// TIA Portal V17 export
// export: Created 2025-01-08T13:55:31.8080412Z, ExportSetting WithDefaults, DisplayName Totally Integrated Automation Portal, DisplayVersion V17, DisplayName TIA Portal Openness, DisplayVersion V17, DisplayName TIA Portal Version Control Interface, DisplayVersion V17, DisplayName SINAMICS Startdrive Advanced, DisplayVersion V17 Update2, DisplayName SINAMICS Startdrive G130, G150, S120, S150, SINAMICS MV, S210, DisplayVersion V17 Update2, DisplayName SINAMICS Startdrive G110M, G120, G120C, G120D, G120P, G115D, DisplayVersion V17 Update2, DisplayName STEP 7 Professional, DisplayVersion V17, DisplayName STEP 7 Safety, DisplayVersion V17, DisplayName WinCC Advanced, DisplayVersion V17
FUNCTION_BLOCK "FB_Com"   // FB1, LAD
{ S7_Optimized_Access := 'TRUE' }
VERSION : 0.1
// stored: AutoNumber true, IsIECCheckEnabled false, IsRetainMemResEnabled false, MemoryReserve 100, SetENOAutomatically false, UDAEnableTagReadback false
   VAR
      TRCV_C_Instance { S7_SetPoint := 'True'} : TRCV_C;
      GET_Instance { S7_SetPoint := 'True'} : GET;
      TRCV_C_Instance_1 { S7_SetPoint := 'True'} : TRCV_C;
      Diff : LInt;
   END_VAR
BEGIN

REGION Network 1
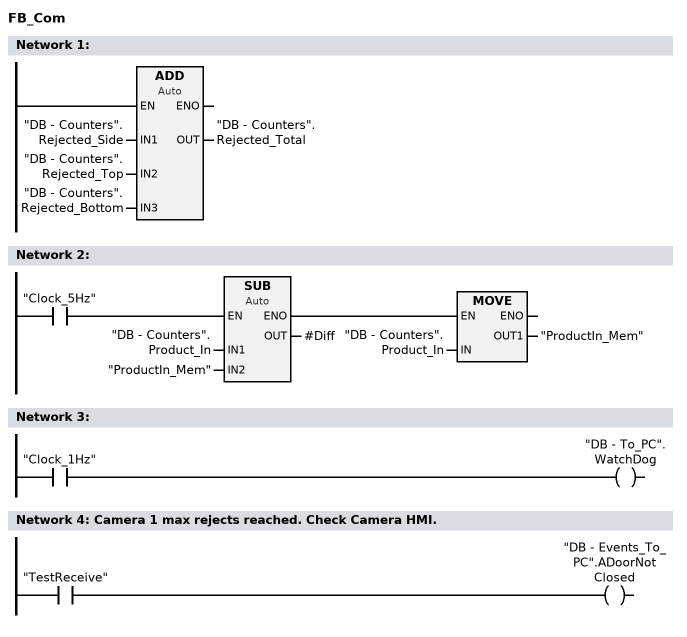
   RUNG wire#powerrail
      Add(in1 := "DB - Counters".Rejected_Side, in2 := "DB - Counters".Rejected_Top, in3 := "DB - Counters".Rejected_Bottom, out => "DB - Counters".Rejected_Total)
   END_RUNG
   // the same network as SCL:
   "DB - Counters".Rejected_Total := "DB - Counters".Rejected_Side + "DB - Counters".Rejected_Top + "DB - Counters".Rejected_Bottom;
END_REGION

REGION Network 2
   RUNG wire#powerrail
      Contact( "Clock_5Hz" )
      Sub(in1 := "DB - Counters".Product_In, in2 := "ProductIn_Mem", out => #Diff)
      Move(in := "DB - Counters".Product_In, out1 => "ProductIn_Mem")
   END_RUNG
   // the same network as SCL:
   IF "Clock_5Hz" THEN
       #Diff := "DB - Counters".Product_In - "ProductIn_Mem";
       "ProductIn_Mem" := "DB - Counters".Product_In;
   END_IF;
END_REGION

REGION Network 3
   RUNG wire#powerrail
      Contact( "Clock_1Hz" )
      Coil( "DB - To_PC".WatchDog )
   END_RUNG
   // the same network as SCL:
   "DB - To_PC".WatchDog := "Clock_1Hz";
END_REGION

REGION Network 4: Camera 1 max rejects reached. Check Camera HMI.
   RUNG wire#powerrail
      Contact( "TestReceive" )
      Coil( "DB - Events_To_PC".ADoorNotClosed )
   END_RUNG
   // the same network as SCL:
   "DB - Events_To_PC".ADoorNotClosed := "TestReceive";
END_REGION
END_FUNCTION_BLOCK
